(* Common base of all reusable behavior types. *)
FUNCTION_BLOCK ABSTRACT BehaviorBase
VAR_INPUT
	i_params: ParameterSet;
END_VAR
VAR_OUTPUT
	{attribute 'OPC.UA.DA' := '1'}
	{attribute 'OPC.UA.DA.Access' := '1'}
	o_status: EOperationResult;
END_VAR
VAR
	(* Because all Control Primitives and Module Sequences instances are 
       singletons, they can set their IDs themselves *)
	{attribute 'OPC.UA.DA' := '1'}
	{attribute 'OPC.UA.DA.Access' := '1'}
	m_id: UINT;
	
	(* define's the behavior's parameters (if any)
	   format: <Name1>:<Type1>;<Name2>:<Type2>;... *)
	{attribute 'OPC.UA.DA' := '1'}
	{attribute 'OPC.UA.DA.Access' := '1'}
	m_paramDefinition: STRING;
END_VAR

PROPERTY Id : UINT
GET
Id := m_id;
END_GET
END_PROPERTY

PROPERTY ABSTRACT Postcondition : IExpression
GET
END_GET
END_PROPERTY

PROPERTY ABSTRACT Precondition : IExpression
GET
END_GET
END_PROPERTY

END_FUNCTION_BLOCK

(* stored: Version 1.1.0.1
   POU BehaviorBase: Id {9d4d1066-c534-403d-9661-100da8d2681e}, SpecialFunc None
   Property Id: Id {ba153d7e-7756-45e1-b8e0-5f9e442e030a}
   Get Get: Id {981a86db-813a-4131-b3fb-fb631a3fc35e}
   Property Postcondition: Id {90225cfd-13e1-444c-bc8a-323cf6976b8b}
   Get Get: Id {b041eb4c-ce04-48b4-94bd-b361fefbcea0}
   Property Precondition: Id {628feb89-8bb5-47be-9aa3-63217f9f17f7}
   Get Get: Id {b908d781-8451-454e-b15f-ef2782e48345} *)
